// TwinCAT 3 PLC project PLC
// Title: Tc3Build Library
// Company: Tc3Build
// ProjectVersion: 1.0.0.0
// ProgramVersion: 3.1.4026.27
// libraries:
//   Tc2_Standard, * (Beckhoff Automation GmbH)
//   Tc2_System, * (Beckhoff Automation GmbH)
// project tree:
//   / PlcTask.TcTTO
//   POUs/ MAIN.TcPOU

CONFIGURATION PLC
    RESOURCE PLC ON TwinCAT3
        TASK PlcTask(INTERVAL := T#10ms, PRIORITY := 20);
        PROGRAM MAIN WITH PlcTask : MAIN;
    END_RESOURCE
END_CONFIGURATION

// ---- POUs/MAIN.TcPOU
PROGRAM MAIN
VAR
	_Count			: UINT;
END_VAR

_Count := _Count + 1;

END_PROGRAM
